// TIA Portal V17 export
// export: Created 2025-03-12T15:34:11.8614261Z, ExportSetting WithDefaults, DisplayName Totally Integrated Automation Portal, DisplayVersion V17 Update 8, DisplayName TIA Portal Openness, DisplayVersion V17 Update 8, DisplayName TIA Portal Version Control Interface, DisplayVersion V17, DisplayName SINAMICS Startdrive Advanced, DisplayVersion V17 SP2, DisplayName SINAMICS Startdrive G110M, G120, G120C, G120D, G120P, G115D, DisplayVersion V17 SP2, DisplayName SINAMICS Startdrive G130, G150, S120, S150, SINAMICS MV, S210, DisplayVersion V17 SP2, DisplayName STEP 7 Professional, DisplayVersion V17 Update 8, DisplayName SINUMERIK ONE STEP 7 Toolbox, DisplayVersion V17 Update 12, DisplayName SINUMERIK 840D sl STEP 7 Toolbox, DisplayVersion V17 Update 12, DisplayName STEP 7 Safety, DisplayVersion V17 Update 6, DisplayName WinCC Advanced, DisplayVersion V17 Update 8
FUNCTION "FC1452_AUXILIARY_COOLING_SYSTEM" : Void   // FC1452, LAD
{ S7_Optimized_Access := 'TRUE' }
VERSION : 0.1
// stored: AutoNumber false, IsIECCheckEnabled false, SetENOAutomatically false, UDAEnableTagReadback false
   VAR_TEMP
      FLOW_AUX : Real;
      TEMPERATURE_AUX : Int;
   END_VAR
BEGIN

REGION Network 1: <<<<<<<<<<<< SHIELD COOLING SYSTEM UNITS 01 & 02>>>>>>>>>>>>>>>>>>>
END_REGION

REGION Network 2: CALL FB1452 SHIELD AUXILIARY COOLING SYSTEM
   // 2#0000_0001 OPTIONS 0 BIT 0 GENERAL CIRCUIT BRAKER ALARM
   // 2#0000_0010 OPTIONS 0 BIT 1 GENERAL CONTACTOR FEEDBACK ALARM
   // 2#0000_0100 OPTIONS 0 BIT 2 UNIT 01 FLOW SETPOINT ALARM
   // 2#0000_1000 OPTIONS 0 BIT 3 UNIT 01 TEMPERATURE SETPOINT ALARM
   // 2#0001_0000 OPTIONS 0 BIT 4 SPARE
   // 2#0010_0000 OPTIONS 0 BIT 5 SPARE
   // 2#0100_0000 OPTIONS 0 BIT 6 SPARE
   // 2#1000_0000 OPTIONS 0 BIT 7 SPARE
   // 
   // 2#0000_0001 OPTIONS 1 BIT 0 FIRST FEEDBACK FLOW TEMPERATURE SENSOR (UNIT 01)
   // 2#0000_0010 OPTIONS 1 BIT 1 SECOND FEEDBACK FLOW TEMPERATURE SENSOR (UNIT 02)
   // 2#0000_0100 OPTIONS 1 BIT 2 UNIT 02 FLOW SETPOINT ALARM
   // 2#0000_1000 OPTIONS 1 BIT 3 UNIT 02 TEMPERATURE SETPOINT ALARM
   // 2#0001_0000 OPTIONS 1 BIT 4 SPARE
   // 2#0010_0000 OPTIONS 1 BIT 5 SPARE
   // 2#0100_0000 OPTIONS 1 BIT 6 SPARE
   // 2#1000_0000 OPTIONS 1 BIT 7 SPARE
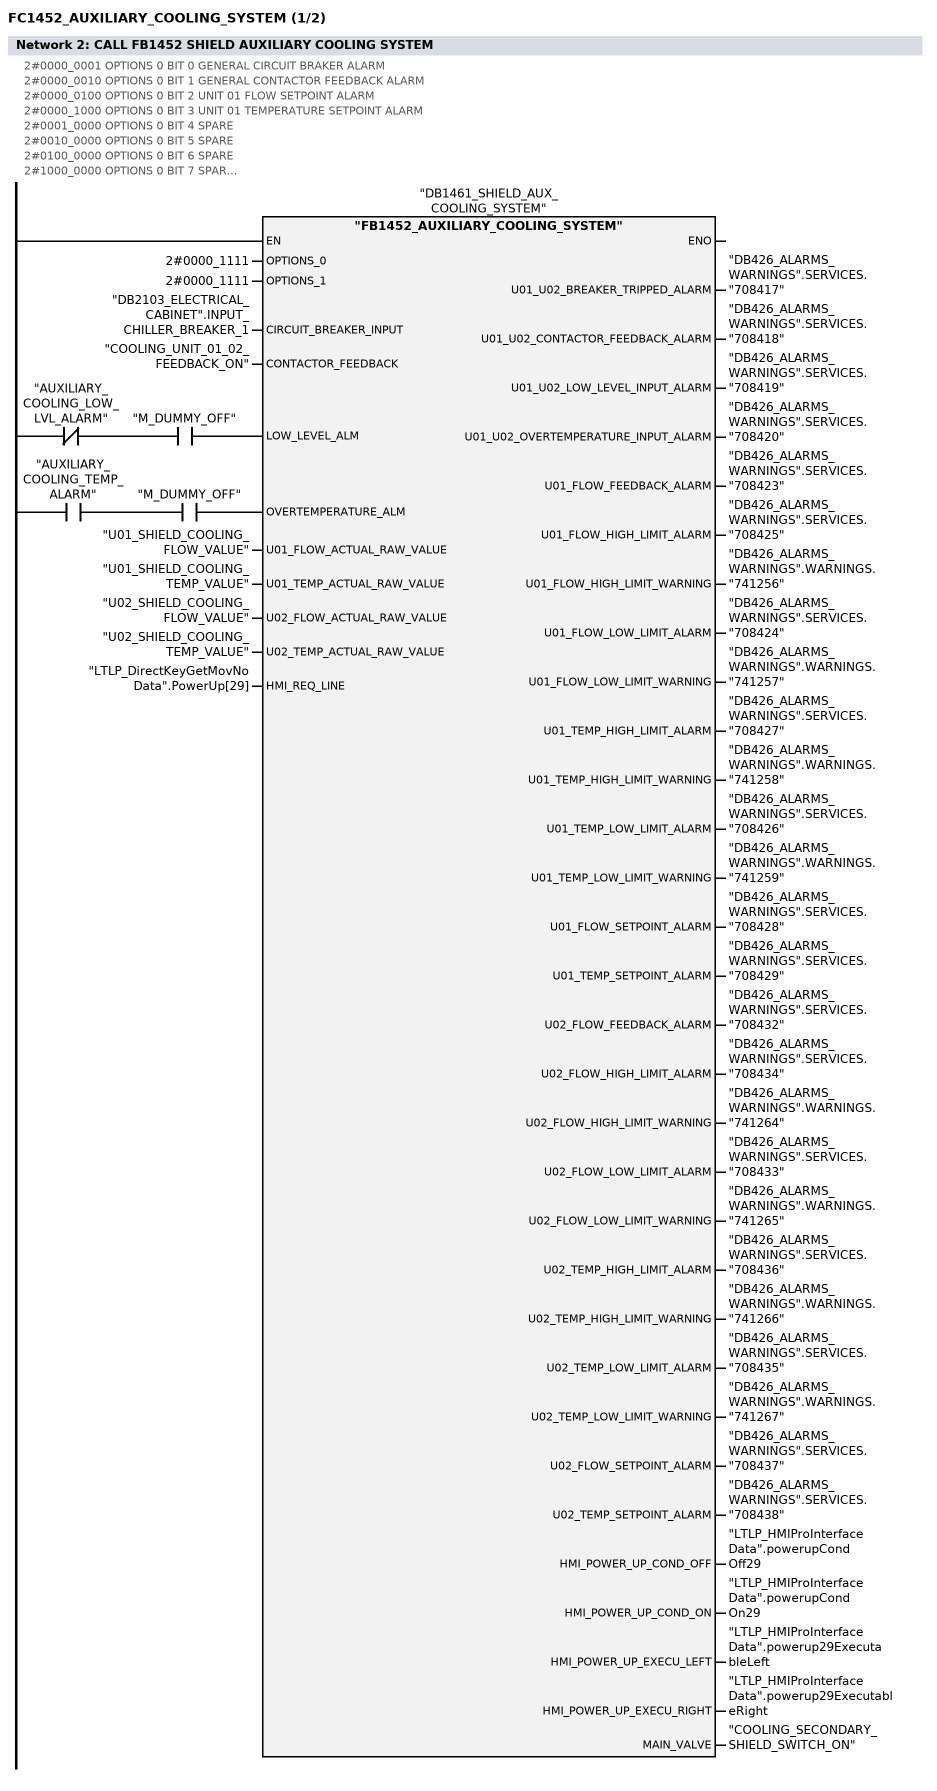
   RUNG wire#powerrail
      "DB1461_SHIELD_AUX_COOLING_SYSTEM"(LOW_LEVEL_ALM := wire#w1, OVERTEMPERATURE_ALM := wire#w2, OPTIONS_0 := 2#0000_1111, OPTIONS_1 := 2#0000_1111, CIRCUIT_BREAKER_INPUT := "DB2103_ELECTRICAL_CABINET".INPUT_CHILLER_BREAKER_1, CONTACTOR_FEEDBACK := "COOLING_UNIT_01_02_FEEDBACK_ON", U01_FLOW_ACTUAL_RAW_VALUE := "U01_SHIELD_COOLING_FLOW_VALUE", U01_TEMP_ACTUAL_RAW_VALUE := "U01_SHIELD_COOLING_TEMP_VALUE", U02_FLOW_ACTUAL_RAW_VALUE := "U02_SHIELD_COOLING_FLOW_VALUE", U02_TEMP_ACTUAL_RAW_VALUE := "U02_SHIELD_COOLING_TEMP_VALUE", HMI_REQ_LINE := "LTLP_DirectKeyGetMovNoData".PowerUp[29], U01_U02_BREAKER_TRIPPED_ALARM => "DB426_ALARMS_WARNINGS".SERVICES."708417", U01_U02_CONTACTOR_FEEDBACK_ALARM => "DB426_ALARMS_WARNINGS".SERVICES."708418", U01_U02_LOW_LEVEL_INPUT_ALARM => "DB426_ALARMS_WARNINGS".SERVICES."708419", U01_U02_OVERTEMPERATURE_INPUT_ALARM => "DB426_ALARMS_WARNINGS".SERVICES."708420", U01_FLOW_FEEDBACK_ALARM => "DB426_ALARMS_WARNINGS".SERVICES."708423", U01_FLOW_HIGH_LIMIT_ALARM => "DB426_ALARMS_WARNINGS".SERVICES."708425", U01_FLOW_HIGH_LIMIT_WARNING => "DB426_ALARMS_WARNINGS".WARNINGS."741256", U01_FLOW_LOW_LIMIT_ALARM => "DB426_ALARMS_WARNINGS".SERVICES."708424", U01_FLOW_LOW_LIMIT_WARNING => "DB426_ALARMS_WARNINGS".WARNINGS."741257", U01_TEMP_HIGH_LIMIT_ALARM => "DB426_ALARMS_WARNINGS".SERVICES."708427", U01_TEMP_HIGH_LIMIT_WARNING => "DB426_ALARMS_WARNINGS".WARNINGS."741258", U01_TEMP_LOW_LIMIT_ALARM => "DB426_ALARMS_WARNINGS".SERVICES."708426", U01_TEMP_LOW_LIMIT_WARNING => "DB426_ALARMS_WARNINGS".WARNINGS."741259", U01_FLOW_SETPOINT_ALARM => "DB426_ALARMS_WARNINGS".SERVICES."708428", U01_TEMP_SETPOINT_ALARM => "DB426_ALARMS_WARNINGS".SERVICES."708429", U02_FLOW_FEEDBACK_ALARM => "DB426_ALARMS_WARNINGS".SERVICES."708432", U02_FLOW_HIGH_LIMIT_ALARM => "DB426_ALARMS_WARNINGS".SERVICES."708434", U02_FLOW_HIGH_LIMIT_WARNING => "DB426_ALARMS_WARNINGS".WARNINGS."741264", U02_FLOW_LOW_LIMIT_ALARM => "DB426_ALARMS_WARNINGS".SERVICES."708433", U02_FLOW_LOW_LIMIT_WARNING => "DB426_ALARMS_WARNINGS".WARNINGS."741265", U02_TEMP_HIGH_LIMIT_ALARM => "DB426_ALARMS_WARNINGS".SERVICES."708436", U02_TEMP_HIGH_LIMIT_WARNING => "DB426_ALARMS_WARNINGS".WARNINGS."741266", U02_TEMP_LOW_LIMIT_ALARM => "DB426_ALARMS_WARNINGS".SERVICES."708435", U02_TEMP_LOW_LIMIT_WARNING => "DB426_ALARMS_WARNINGS".WARNINGS."741267", U02_FLOW_SETPOINT_ALARM => "DB426_ALARMS_WARNINGS".SERVICES."708437", U02_TEMP_SETPOINT_ALARM => "DB426_ALARMS_WARNINGS".SERVICES."708438", HMI_POWER_UP_COND_OFF => "LTLP_HMIProInterfaceData".powerupCondOff29, HMI_POWER_UP_COND_ON => "LTLP_HMIProInterfaceData".powerupCondOn29, HMI_POWER_UP_EXECU_LEFT => "LTLP_HMIProInterfaceData".powerup29ExecutableLeft, HMI_POWER_UP_EXECU_RIGHT => "LTLP_HMIProInterfaceData".powerup29ExecutableRight, MAIN_VALVE => "COOLING_SECONDARY_SHIELD_SWITCH_ON")
   END_RUNG
   RUNG wire#powerrail
      I_Contact( "AUXILIARY_COOLING_LOW_LVL_ALARM" )
      Contact( "M_DUMMY_OFF" )
   END_RUNG wire#w1
   RUNG wire#powerrail
      Contact( "AUXILIARY_COOLING_TEMP_ALARM" )
      Contact( "M_DUMMY_OFF" )
   END_RUNG wire#w2
   // the same network as SCL:
   "DB1461_SHIELD_AUX_COOLING_SYSTEM"(OPTIONS_0 := 2#0000_1111,   // "FB1452_AUXILIARY_COOLING_SYSTEM"
                           OPTIONS_1 := 2#0000_1111,
                           CIRCUIT_BREAKER_INPUT := "DB2103_ELECTRICAL_CABINET".INPUT_CHILLER_BREAKER_1,
                           CONTACTOR_FEEDBACK := "COOLING_UNIT_01_02_FEEDBACK_ON",
                           LOW_LEVEL_ALM := NOT "AUXILIARY_COOLING_LOW_LVL_ALARM" AND "M_DUMMY_OFF",
                           OVERTEMPERATURE_ALM := "AUXILIARY_COOLING_TEMP_ALARM" AND "M_DUMMY_OFF",
                           U01_FLOW_ACTUAL_RAW_VALUE := "U01_SHIELD_COOLING_FLOW_VALUE",
                           U01_TEMP_ACTUAL_RAW_VALUE := "U01_SHIELD_COOLING_TEMP_VALUE",
                           U02_FLOW_ACTUAL_RAW_VALUE := "U02_SHIELD_COOLING_FLOW_VALUE",
                           U02_TEMP_ACTUAL_RAW_VALUE := "U02_SHIELD_COOLING_TEMP_VALUE",
                           HMI_REQ_LINE := "LTLP_DirectKeyGetMovNoData".PowerUp[29],
                           U01_U02_BREAKER_TRIPPED_ALARM => "DB426_ALARMS_WARNINGS".SERVICES."708417",
                           U01_U02_CONTACTOR_FEEDBACK_ALARM => "DB426_ALARMS_WARNINGS".SERVICES."708418",
                           U01_U02_LOW_LEVEL_INPUT_ALARM => "DB426_ALARMS_WARNINGS".SERVICES."708419",
                           U01_U02_OVERTEMPERATURE_INPUT_ALARM => "DB426_ALARMS_WARNINGS".SERVICES."708420",
                           U01_FLOW_FEEDBACK_ALARM => "DB426_ALARMS_WARNINGS".SERVICES."708423",
                           U01_FLOW_HIGH_LIMIT_ALARM => "DB426_ALARMS_WARNINGS".SERVICES."708425",
                           U01_FLOW_HIGH_LIMIT_WARNING => "DB426_ALARMS_WARNINGS".WARNINGS."741256",
                           U01_FLOW_LOW_LIMIT_ALARM => "DB426_ALARMS_WARNINGS".SERVICES."708424",
                           U01_FLOW_LOW_LIMIT_WARNING => "DB426_ALARMS_WARNINGS".WARNINGS."741257",
                           U01_TEMP_HIGH_LIMIT_ALARM => "DB426_ALARMS_WARNINGS".SERVICES."708427",
                           U01_TEMP_HIGH_LIMIT_WARNING => "DB426_ALARMS_WARNINGS".WARNINGS."741258",
                           U01_TEMP_LOW_LIMIT_ALARM => "DB426_ALARMS_WARNINGS".SERVICES."708426",
                           U01_TEMP_LOW_LIMIT_WARNING => "DB426_ALARMS_WARNINGS".WARNINGS."741259",
                           U01_FLOW_SETPOINT_ALARM => "DB426_ALARMS_WARNINGS".SERVICES."708428",
                           U01_TEMP_SETPOINT_ALARM => "DB426_ALARMS_WARNINGS".SERVICES."708429",
                           U02_FLOW_FEEDBACK_ALARM => "DB426_ALARMS_WARNINGS".SERVICES."708432",
                           U02_FLOW_HIGH_LIMIT_ALARM => "DB426_ALARMS_WARNINGS".SERVICES."708434",
                           U02_FLOW_HIGH_LIMIT_WARNING => "DB426_ALARMS_WARNINGS".WARNINGS."741264",
                           U02_FLOW_LOW_LIMIT_ALARM => "DB426_ALARMS_WARNINGS".SERVICES."708433",
                           U02_FLOW_LOW_LIMIT_WARNING => "DB426_ALARMS_WARNINGS".WARNINGS."741265",
                           U02_TEMP_HIGH_LIMIT_ALARM => "DB426_ALARMS_WARNINGS".SERVICES."708436",
                           U02_TEMP_HIGH_LIMIT_WARNING => "DB426_ALARMS_WARNINGS".WARNINGS."741266",
                           U02_TEMP_LOW_LIMIT_ALARM => "DB426_ALARMS_WARNINGS".SERVICES."708435",
                           U02_TEMP_LOW_LIMIT_WARNING => "DB426_ALARMS_WARNINGS".WARNINGS."741267",
                           U02_FLOW_SETPOINT_ALARM => "DB426_ALARMS_WARNINGS".SERVICES."708437",
                           U02_TEMP_SETPOINT_ALARM => "DB426_ALARMS_WARNINGS".SERVICES."708438",
                           HMI_POWER_UP_COND_OFF => "LTLP_HMIProInterfaceData".powerupCondOff29,
                           HMI_POWER_UP_COND_ON => "LTLP_HMIProInterfaceData".powerupCondOn29,
                           HMI_POWER_UP_EXECU_LEFT => "LTLP_HMIProInterfaceData".powerup29ExecutableLeft,
                           HMI_POWER_UP_EXECU_RIGHT => "LTLP_HMIProInterfaceData".powerup29ExecutableRight,
                           MAIN_VALVE => "COOLING_SECONDARY_SHIELD_SWITCH_ON");
END_REGION

REGION Network 3: CALL FB1452 CELL COOLING BUFFER AUXILIARY COOLING SYSTEM
   // 2#0000_0001 OPTIONS 0 BIT 0 GENERAL CIRCUIT BRAKER ALARM
   // 2#0000_0010 OPTIONS 0 BIT 1 GENERAL CONTACTOR FEEDBACK ALARM
   // 2#0000_0100 OPTIONS 0 BIT 2 UNIT 01 FLOW SETPOINT ALARM
   // 2#0000_1000 OPTIONS 0 BIT 3 UNIT 01 TEMPERATURE SETPOINT ALARM
   // 2#0001_0000 OPTIONS 0 BIT 4 SPARE
   // 2#0010_0000 OPTIONS 0 BIT 5 SPARE
   // 2#0100_0000 OPTIONS 0 BIT 6 SPARE
   // 2#1000_0000 OPTIONS 0 BIT 7 SPARE
   // 
   // 2#0000_0001 OPTIONS 1 BIT 0 FIRST FEEDBACK FLOW TEMPERATURE SENSOR (UNIT 01)
   // 2#0000_0010 OPTIONS 1 BIT 1 SECOND FEEDBACK FLOW TEMPERATURE SENSOR (UNIT 02)
   // 2#0000_0100 OPTIONS 1 BIT 2 UNIT 02 FLOW SETPOINT ALARM
   // 2#0000_1000 OPTIONS 1 BIT 3 UNIT 02 TEMPERATURE SETPOINT ALARM
   // 2#0001_0000 OPTIONS 1 BIT 4 SPARE
   // 2#0010_0000 OPTIONS 1 BIT 5 SPARE
   // 2#0100_0000 OPTIONS 1 BIT 6 SPARE
   // 2#1000_0000 OPTIONS 1 BIT 7 SPARE
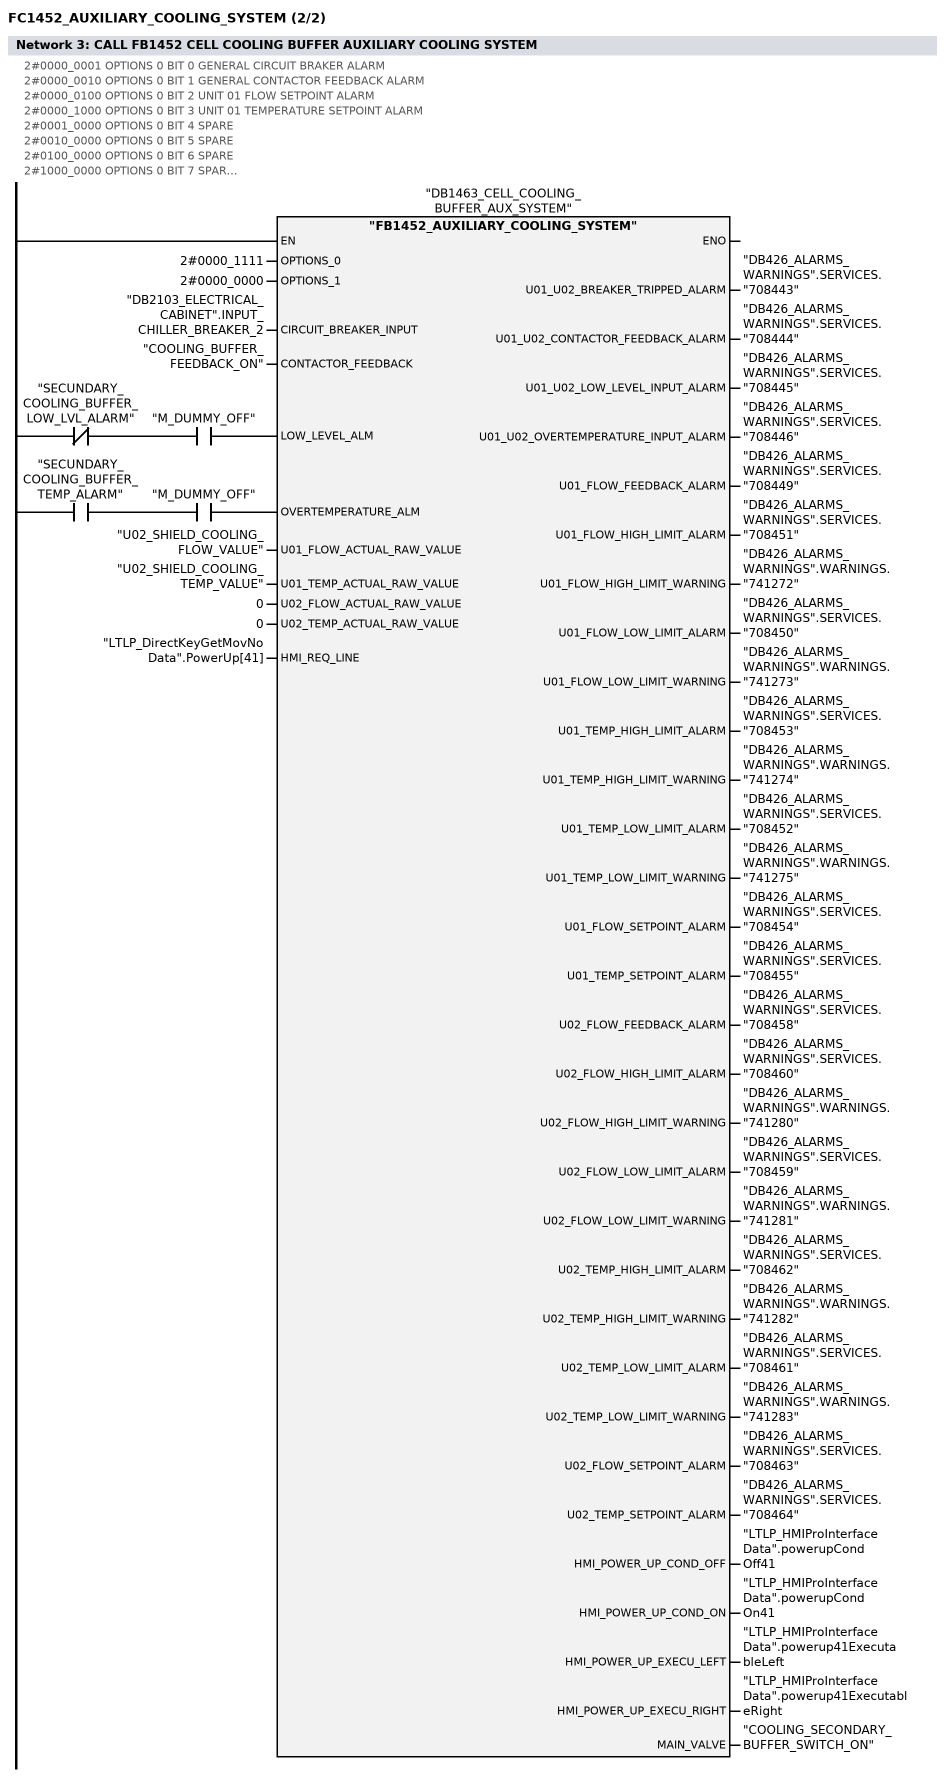
   RUNG wire#powerrail
      "DB1463_CELL_COOLING_BUFFER_AUX_SYSTEM"(LOW_LEVEL_ALM := wire#w1, OVERTEMPERATURE_ALM := wire#w2, OPTIONS_0 := 2#0000_1111, OPTIONS_1 := 2#0000_0000, CIRCUIT_BREAKER_INPUT := "DB2103_ELECTRICAL_CABINET".INPUT_CHILLER_BREAKER_2, CONTACTOR_FEEDBACK := "COOLING_BUFFER_FEEDBACK_ON", U01_FLOW_ACTUAL_RAW_VALUE := "U02_SHIELD_COOLING_FLOW_VALUE", U01_TEMP_ACTUAL_RAW_VALUE := "U02_SHIELD_COOLING_TEMP_VALUE", U02_FLOW_ACTUAL_RAW_VALUE := 0, U02_TEMP_ACTUAL_RAW_VALUE := 0, HMI_REQ_LINE := "LTLP_DirectKeyGetMovNoData".PowerUp[41], U01_U02_BREAKER_TRIPPED_ALARM => "DB426_ALARMS_WARNINGS".SERVICES."708443", U01_U02_CONTACTOR_FEEDBACK_ALARM => "DB426_ALARMS_WARNINGS".SERVICES."708444", U01_U02_LOW_LEVEL_INPUT_ALARM => "DB426_ALARMS_WARNINGS".SERVICES."708445", U01_U02_OVERTEMPERATURE_INPUT_ALARM => "DB426_ALARMS_WARNINGS".SERVICES."708446", U01_FLOW_FEEDBACK_ALARM => "DB426_ALARMS_WARNINGS".SERVICES."708449", U01_FLOW_HIGH_LIMIT_ALARM => "DB426_ALARMS_WARNINGS".SERVICES."708451", U01_FLOW_HIGH_LIMIT_WARNING => "DB426_ALARMS_WARNINGS".WARNINGS."741272", U01_FLOW_LOW_LIMIT_ALARM => "DB426_ALARMS_WARNINGS".SERVICES."708450", U01_FLOW_LOW_LIMIT_WARNING => "DB426_ALARMS_WARNINGS".WARNINGS."741273", U01_TEMP_HIGH_LIMIT_ALARM => "DB426_ALARMS_WARNINGS".SERVICES."708453", U01_TEMP_HIGH_LIMIT_WARNING => "DB426_ALARMS_WARNINGS".WARNINGS."741274", U01_TEMP_LOW_LIMIT_ALARM => "DB426_ALARMS_WARNINGS".SERVICES."708452", U01_TEMP_LOW_LIMIT_WARNING => "DB426_ALARMS_WARNINGS".WARNINGS."741275", U01_FLOW_SETPOINT_ALARM => "DB426_ALARMS_WARNINGS".SERVICES."708454", U01_TEMP_SETPOINT_ALARM => "DB426_ALARMS_WARNINGS".SERVICES."708455", U02_FLOW_FEEDBACK_ALARM => "DB426_ALARMS_WARNINGS".SERVICES."708458", U02_FLOW_HIGH_LIMIT_ALARM => "DB426_ALARMS_WARNINGS".SERVICES."708460", U02_FLOW_HIGH_LIMIT_WARNING => "DB426_ALARMS_WARNINGS".WARNINGS."741280", U02_FLOW_LOW_LIMIT_ALARM => "DB426_ALARMS_WARNINGS".SERVICES."708459", U02_FLOW_LOW_LIMIT_WARNING => "DB426_ALARMS_WARNINGS".WARNINGS."741281", U02_TEMP_HIGH_LIMIT_ALARM => "DB426_ALARMS_WARNINGS".SERVICES."708462", U02_TEMP_HIGH_LIMIT_WARNING => "DB426_ALARMS_WARNINGS".WARNINGS."741282", U02_TEMP_LOW_LIMIT_ALARM => "DB426_ALARMS_WARNINGS".SERVICES."708461", U02_TEMP_LOW_LIMIT_WARNING => "DB426_ALARMS_WARNINGS".WARNINGS."741283", U02_FLOW_SETPOINT_ALARM => "DB426_ALARMS_WARNINGS".SERVICES."708463", U02_TEMP_SETPOINT_ALARM => "DB426_ALARMS_WARNINGS".SERVICES."708464", HMI_POWER_UP_COND_OFF => "LTLP_HMIProInterfaceData".powerupCondOff41, HMI_POWER_UP_COND_ON => "LTLP_HMIProInterfaceData".powerupCondOn41, HMI_POWER_UP_EXECU_LEFT => "LTLP_HMIProInterfaceData".powerup41ExecutableLeft, HMI_POWER_UP_EXECU_RIGHT => "LTLP_HMIProInterfaceData".powerup41ExecutableRight, MAIN_VALVE => "COOLING_SECONDARY_BUFFER_SWITCH_ON")
   END_RUNG
   RUNG wire#powerrail
      I_Contact( "SECUNDARY_COOLING_BUFFER_LOW_LVL_ALARM" )
      Contact( "M_DUMMY_OFF" )
   END_RUNG wire#w1
   RUNG wire#powerrail
      Contact( "SECUNDARY_COOLING_BUFFER_TEMP_ALARM" )
      Contact( "M_DUMMY_OFF" )
   END_RUNG wire#w2
   // the same network as SCL:
   "DB1463_CELL_COOLING_BUFFER_AUX_SYSTEM"(OPTIONS_0 := 2#0000_1111,   // "FB1452_AUXILIARY_COOLING_SYSTEM"
                           OPTIONS_1 := 2#0000_0000,
                           CIRCUIT_BREAKER_INPUT := "DB2103_ELECTRICAL_CABINET".INPUT_CHILLER_BREAKER_2,
                           CONTACTOR_FEEDBACK := "COOLING_BUFFER_FEEDBACK_ON",
                           LOW_LEVEL_ALM := NOT "SECUNDARY_COOLING_BUFFER_LOW_LVL_ALARM" AND "M_DUMMY_OFF",
                           OVERTEMPERATURE_ALM := "SECUNDARY_COOLING_BUFFER_TEMP_ALARM" AND "M_DUMMY_OFF",
                           U01_FLOW_ACTUAL_RAW_VALUE := "U02_SHIELD_COOLING_FLOW_VALUE",
                           U01_TEMP_ACTUAL_RAW_VALUE := "U02_SHIELD_COOLING_TEMP_VALUE",
                           U02_FLOW_ACTUAL_RAW_VALUE := 0,
                           U02_TEMP_ACTUAL_RAW_VALUE := 0,
                           HMI_REQ_LINE := "LTLP_DirectKeyGetMovNoData".PowerUp[41],
                           U01_U02_BREAKER_TRIPPED_ALARM => "DB426_ALARMS_WARNINGS".SERVICES."708443",
                           U01_U02_CONTACTOR_FEEDBACK_ALARM => "DB426_ALARMS_WARNINGS".SERVICES."708444",
                           U01_U02_LOW_LEVEL_INPUT_ALARM => "DB426_ALARMS_WARNINGS".SERVICES."708445",
                           U01_U02_OVERTEMPERATURE_INPUT_ALARM => "DB426_ALARMS_WARNINGS".SERVICES."708446",
                           U01_FLOW_FEEDBACK_ALARM => "DB426_ALARMS_WARNINGS".SERVICES."708449",
                           U01_FLOW_HIGH_LIMIT_ALARM => "DB426_ALARMS_WARNINGS".SERVICES."708451",
                           U01_FLOW_HIGH_LIMIT_WARNING => "DB426_ALARMS_WARNINGS".WARNINGS."741272",
                           U01_FLOW_LOW_LIMIT_ALARM => "DB426_ALARMS_WARNINGS".SERVICES."708450",
                           U01_FLOW_LOW_LIMIT_WARNING => "DB426_ALARMS_WARNINGS".WARNINGS."741273",
                           U01_TEMP_HIGH_LIMIT_ALARM => "DB426_ALARMS_WARNINGS".SERVICES."708453",
                           U01_TEMP_HIGH_LIMIT_WARNING => "DB426_ALARMS_WARNINGS".WARNINGS."741274",
                           U01_TEMP_LOW_LIMIT_ALARM => "DB426_ALARMS_WARNINGS".SERVICES."708452",
                           U01_TEMP_LOW_LIMIT_WARNING => "DB426_ALARMS_WARNINGS".WARNINGS."741275",
                           U01_FLOW_SETPOINT_ALARM => "DB426_ALARMS_WARNINGS".SERVICES."708454",
                           U01_TEMP_SETPOINT_ALARM => "DB426_ALARMS_WARNINGS".SERVICES."708455",
                           U02_FLOW_FEEDBACK_ALARM => "DB426_ALARMS_WARNINGS".SERVICES."708458",
                           U02_FLOW_HIGH_LIMIT_ALARM => "DB426_ALARMS_WARNINGS".SERVICES."708460",
                           U02_FLOW_HIGH_LIMIT_WARNING => "DB426_ALARMS_WARNINGS".WARNINGS."741280",
                           U02_FLOW_LOW_LIMIT_ALARM => "DB426_ALARMS_WARNINGS".SERVICES."708459",
                           U02_FLOW_LOW_LIMIT_WARNING => "DB426_ALARMS_WARNINGS".WARNINGS."741281",
                           U02_TEMP_HIGH_LIMIT_ALARM => "DB426_ALARMS_WARNINGS".SERVICES."708462",
                           U02_TEMP_HIGH_LIMIT_WARNING => "DB426_ALARMS_WARNINGS".WARNINGS."741282",
                           U02_TEMP_LOW_LIMIT_ALARM => "DB426_ALARMS_WARNINGS".SERVICES."708461",
                           U02_TEMP_LOW_LIMIT_WARNING => "DB426_ALARMS_WARNINGS".WARNINGS."741283",
                           U02_FLOW_SETPOINT_ALARM => "DB426_ALARMS_WARNINGS".SERVICES."708463",
                           U02_TEMP_SETPOINT_ALARM => "DB426_ALARMS_WARNINGS".SERVICES."708464",
                           HMI_POWER_UP_COND_OFF => "LTLP_HMIProInterfaceData".powerupCondOff41,
                           HMI_POWER_UP_COND_ON => "LTLP_HMIProInterfaceData".powerupCondOn41,
                           HMI_POWER_UP_EXECU_LEFT => "LTLP_HMIProInterfaceData".powerup41ExecutableLeft,
                           HMI_POWER_UP_EXECU_RIGHT => "LTLP_HMIProInterfaceData".powerup41ExecutableRight,
                           MAIN_VALVE => "COOLING_SECONDARY_BUFFER_SWITCH_ON");
END_REGION
END_FUNCTION
